PROGRAM PRG_TEST
VAR
    fbDataCollectionSequence_Test : FB_DataCollectionSequence_Test;
    fbSystemCalibration_Test : FB_SystemCalibration_Test;
END_VAR


TcUnit.RUN();

END_PROGRAM

(* stored: Version 1.1.0.1
   POU PRG_TEST: Id {d103c899-b7b4-4722-91e3-7518e0de7d91}, SpecialFunc None *)
